TYPE ST_System_HS_Stellwert :
STRUCT
END_STRUCT
END_TYPE

(* stored: Version 1.1.0.1, ProductVersion 3.1.4024.9
   DUT ST_System_HS_Stellwert: Id {f8e1868e-e4f8-4877-84d4-f6a7947b36f9} *)
